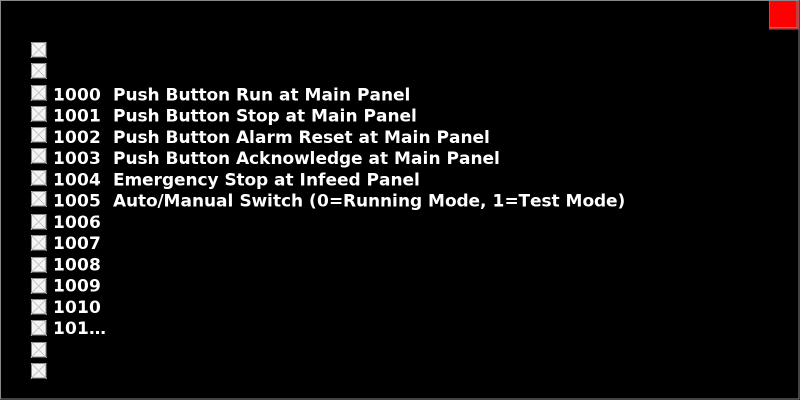
VISUALIZATION P1_DI1  // 800x400, background image 
    ImageSwitcher (31,42 15x15), variable: InputOutput_GVL.xIn1000, behaviour: TOGGLE
    Label (50,16 625x391), "1000 Push Button Run at Main Panel 1001 Push Button Stop at Main Panel 1002 Push Button Alarm Reset at Main Panel 1003 Push Button Acknowledge at Main Panel 1004 Emergency Stop at Infeed Panel 1005 Auto/Manual Switch (0=Running Mode, 1=Test Mode) 1006 1007 1008 1009 1010 1011 1012 1013 1014 1015 Pressure Switch for Main Panel"
    ImageSwitcher (31,63 15x15), variable: InputOutput_GVL.xIn1001, behaviour: TOGGLE
    ImageSwitcher (31,85 15x15), variable: InputOutput_GVL.xIn1002, behaviour: TOGGLE
    ImageSwitcher (31,106 15x15), variable: InputOutput_GVL.xIn1003, behaviour: TOGGLE
    ImageSwitcher (31,127 15x15), variable: InputOutput_GVL.xIn1004, behaviour: TOGGLE
    ImageSwitcher (31,148 15x15), variable: InputOutput_GVL.xIn1005, behaviour: TOGGLE
    ImageSwitcher (31,170 15x15), variable: InputOutput_GVL.xIn1006, behaviour: TOGGLE
    ImageSwitcher (31,191 15x15), variable: InputOutput_GVL.xIn1007, behaviour: TOGGLE
    ImageSwitcher (31,214 15x15), variable: InputOutput_GVL.xIn1008, behaviour: TOGGLE
    ImageSwitcher (31,235 15x15), variable: InputOutput_GVL.xIn1009, behaviour: TOGGLE
    ImageSwitcher (31,257 15x15), variable: InputOutput_GVL.xIn1010, behaviour: TOGGLE
    ImageSwitcher (31,278 15x15), variable: InputOutput_GVL.xIn1011, behaviour: TOGGLE
    ImageSwitcher (31,299 15x15), variable: InputOutput_GVL.xIn1012, behaviour: TOGGLE
    ImageSwitcher (31,320 15x15), variable: InputOutput_GVL.xIn1013, behaviour: TOGGLE
    ImageSwitcher (31,342 15x15), variable: InputOutput_GVL.xIn1014, behaviour: TOGGLE
    ImageSwitcher (31,363 15x15), variable: InputOutput_GVL.xIn1015, behaviour: TOGGLE
    Button (769,-1 30x30), image: VisuSymbols.Symbols.Wrong
        OnMouseClick: CloseDialog Dialog=P1_DI1, Result=OK, NumpadKeypadSet=True
END_VISUALIZATION

(* stored: Version 1.1.0.1, ProductVersion 3.1.4024.12
   Visu P1_DI1: Id {115704c1-39bf-4599-9395-ef6c1f88d2ec} *)
